// TIA Portal V21 export
VAR_GLOBAL   // PLC tag table "OutputAnalogici"
   PompaMono_Velocità AT %QW200 : Word;
   PompaPistoni_Velocità AT %QW202 : Word;
   PompaRilancioTorre_Velocità AT %QW204 : Word;
   Contropressione_CP1 AT %QW206 : Word;   // Sicurezza mono pompa pistoni
   Contropressione_CP2 AT %QW208 : Word;   // Fine linea
   Contropressione_CP3 AT %QW210 : Word;   // Fine linea sterilizzatore
   ModulanteRaffreddamentoAcqua_Apertura AT %QW212 : Word;
   ModulanteRiscaldamentoAcqua_Apertura AT %QW214 : Word;
END_VAR
